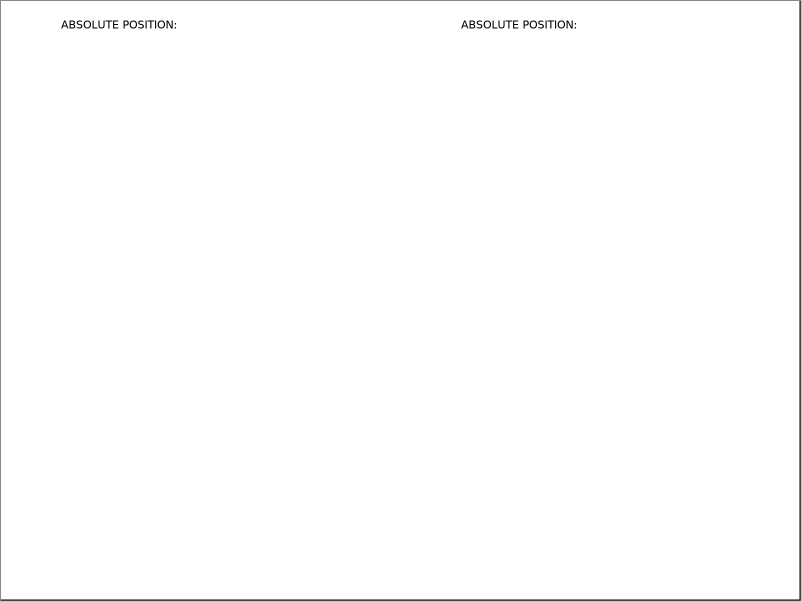
VISUALIZATION F15_Read_Axis_Info  // 802x602
    Rectangle (0,0 800x600)
    Label (10,10 170x30), "ABSOLUTE POSITION:"
    Label (410,10 170x30), "ABSOLUTE POSITION:"
END_VISUALIZATION

(* stored: Version 1.1.0.1, ProductVersion 3.1.4022.7
   Visu F15_Read_Axis_Info: Id {25bf2ca5-1670-469f-a3c8-cc710801c3e5} *)
